// TIA Portal V18 export
// export: Created 2025-12-01T17:51:19.6025932Z, ExportSetting None, DisplayName Totally Integrated Automation Portal, DisplayVersion V18 Update 5, DisplayName TIA Portal Openness, DisplayVersion V18 Update 5, DisplayName TIA Portal Teamcenter Gateway, DisplayVersion V18, DisplayName TIA Portal Version Control Interface, DisplayVersion V18, DisplayName STEP 7 Professional, DisplayVersion V18 Update 5, DisplayName STEP 7 Safety, DisplayVersion V18, DisplayName WinCC Professional, DisplayVersion V18 Update 5
FUNCTION "Motorr" : Void   // FC3100, LAD
{ S7_Optimized_Access := 'TRUE' }
// stored: AutoNumber false, SetENOAutomatically false
   VAR_TEMP   // added for the SCL form of the ladder/FBD networks
      _w1 : Bool;
      _w2 : Bool;
   END_VAR
BEGIN

REGION Network 1: H-shaftLifting_Motor
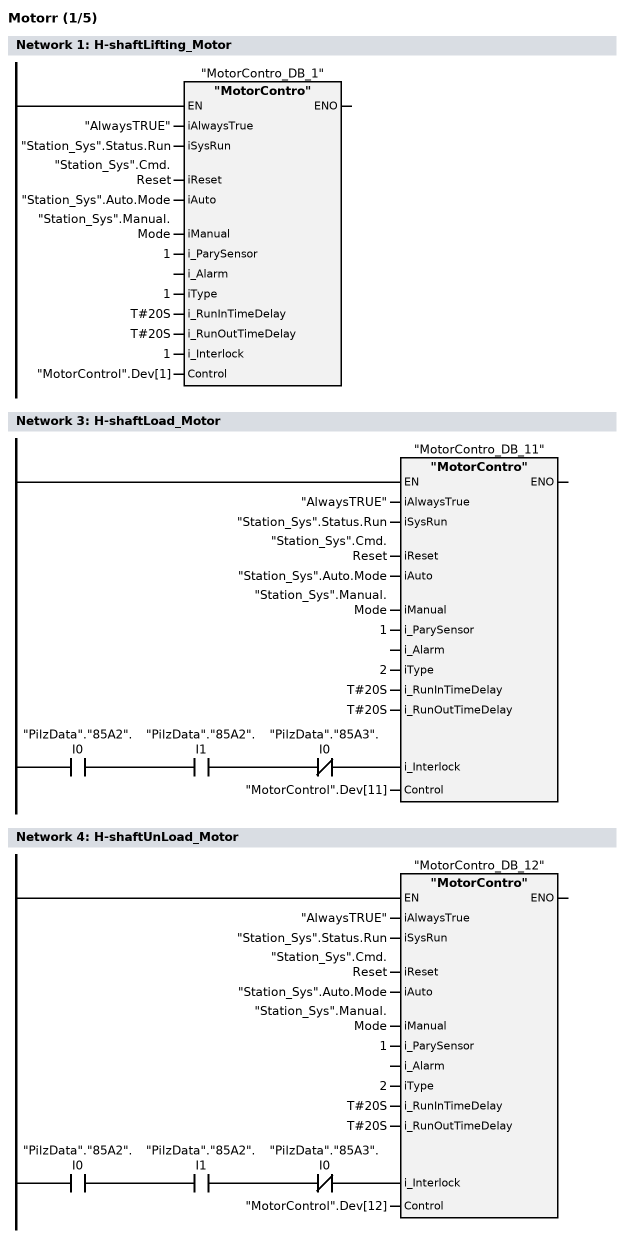
   RUNG wire#powerrail
      "MotorContro_DB_1"(iAlwaysTrue := "AlwaysTRUE", iSysRun := "Station_Sys".Status.Run, iReset := "Station_Sys".Cmd.Reset, iAuto := "Station_Sys".Auto.Mode, iManual := "Station_Sys".Manual.Mode, i_ParySensor := 1, i_Alarm :=, iType := 1, i_RunInTimeDelay := T#20S, i_RunOutTimeDelay := T#20S, i_Interlock := 1, Control := "MotorControl".Dev[1])
   END_RUNG
   // the same network as SCL:
   "MotorContro_DB_1"(iAlwaysTrue := "AlwaysTRUE",   // "MotorContro"
                      iSysRun := "Station_Sys".Status.Run,
                      iReset := "Station_Sys".Cmd.Reset,
                      iAuto := "Station_Sys".Auto.Mode,
                      iManual := "Station_Sys".Manual.Mode,
                      i_ParySensor := 1,
                      iType := 1,
                      i_RunInTimeDelay := T#20S,
                      i_RunOutTimeDelay := T#20S,
                      i_Interlock := 1,
                      Control := "MotorControl".Dev[1]);
END_REGION

REGION Network 2 (SCL): H-shaftLifting_Motor_OutPut
   "oH-shaftLifting_Start" := "MotorControl".Dev[1].OutControl.o_Start;
   "oH-shaftLifting_CCWStart" := "MotorControl".Dev[1].OutControl.o_CCWStart ;
   "oH-shaftLifting_SpeedChange" := "MotorControl".Dev[1].OutControl.o_SpeedChanged;
END_REGION

REGION Network 3: H-shaftLoad_Motor
   RUNG wire#powerrail
      "MotorContro_DB_11"(i_Interlock := wire#w1, iAlwaysTrue := "AlwaysTRUE", iSysRun := "Station_Sys".Status.Run, iReset := "Station_Sys".Cmd.Reset, iAuto := "Station_Sys".Auto.Mode, iManual := "Station_Sys".Manual.Mode, i_ParySensor := 1, i_Alarm :=, iType := 2, i_RunInTimeDelay := T#20S, i_RunOutTimeDelay := T#20S, Control := "MotorControl".Dev[11])
   END_RUNG
   RUNG wire#powerrail
      Contact( "PilzData"."85A2".I0 )
      Contact( "PilzData"."85A2".I1 )
      I_Contact( "PilzData"."85A3".I0 )
   END_RUNG wire#w1
   // the same network as SCL:
   "MotorContro_DB_11"(iAlwaysTrue := "AlwaysTRUE",   // "MotorContro"
                       iSysRun := "Station_Sys".Status.Run,
                       iReset := "Station_Sys".Cmd.Reset,
                       iAuto := "Station_Sys".Auto.Mode,
                       iManual := "Station_Sys".Manual.Mode,
                       i_ParySensor := 1,
                       iType := 2,
                       i_RunInTimeDelay := T#20S,
                       i_RunOutTimeDelay := T#20S,
                       i_Interlock := "PilzData"."85A2".I0 AND "PilzData"."85A2".I1 AND NOT "PilzData"."85A3".I0,
                       Control := "MotorControl".Dev[11]);
END_REGION

REGION Network 4: H-shaftUnLoad_Motor
   RUNG wire#powerrail
      "MotorContro_DB_12"(i_Interlock := wire#w1, iAlwaysTrue := "AlwaysTRUE", iSysRun := "Station_Sys".Status.Run, iReset := "Station_Sys".Cmd.Reset, iAuto := "Station_Sys".Auto.Mode, iManual := "Station_Sys".Manual.Mode, i_ParySensor := 1, i_Alarm :=, iType := 2, i_RunInTimeDelay := T#20S, i_RunOutTimeDelay := T#20S, Control := "MotorControl".Dev[12])
   END_RUNG
   RUNG wire#powerrail
      Contact( "PilzData"."85A2".I0 )
      Contact( "PilzData"."85A2".I1 )
      I_Contact( "PilzData"."85A3".I0 )
   END_RUNG wire#w1
   // the same network as SCL:
   "MotorContro_DB_12"(iAlwaysTrue := "AlwaysTRUE",   // "MotorContro"
                       iSysRun := "Station_Sys".Status.Run,
                       iReset := "Station_Sys".Cmd.Reset,
                       iAuto := "Station_Sys".Auto.Mode,
                       iManual := "Station_Sys".Manual.Mode,
                       i_ParySensor := 1,
                       iType := 2,
                       i_RunInTimeDelay := T#20S,
                       i_RunOutTimeDelay := T#20S,
                       i_Interlock := "PilzData"."85A2".I0 AND "PilzData"."85A2".I1 AND NOT "PilzData"."85A3".I0,
                       Control := "MotorControl".Dev[12]);
END_REGION

REGION Network 5 (SCL): H-shaftLifting_Motor_OutPut / H-shaftLoad_Motor_OutPut
   "oH-shaftLoading_CW" := "MotorControl".Dev[11].OutControl.o_Start;
   "oH-shaftLoading_CCW" := "MotorControl".Dev[11].OutControl.o_CCWStart OR ("Station_Sys".Auto.Mode AND "AutoProcessControl".Global.H.EmptyPallet);

   "oH-shaftTake_CW" := "MotorControl".Dev[12].OutControl.o_Start;
END_REGION

REGION Network 6: Auto MotorStop
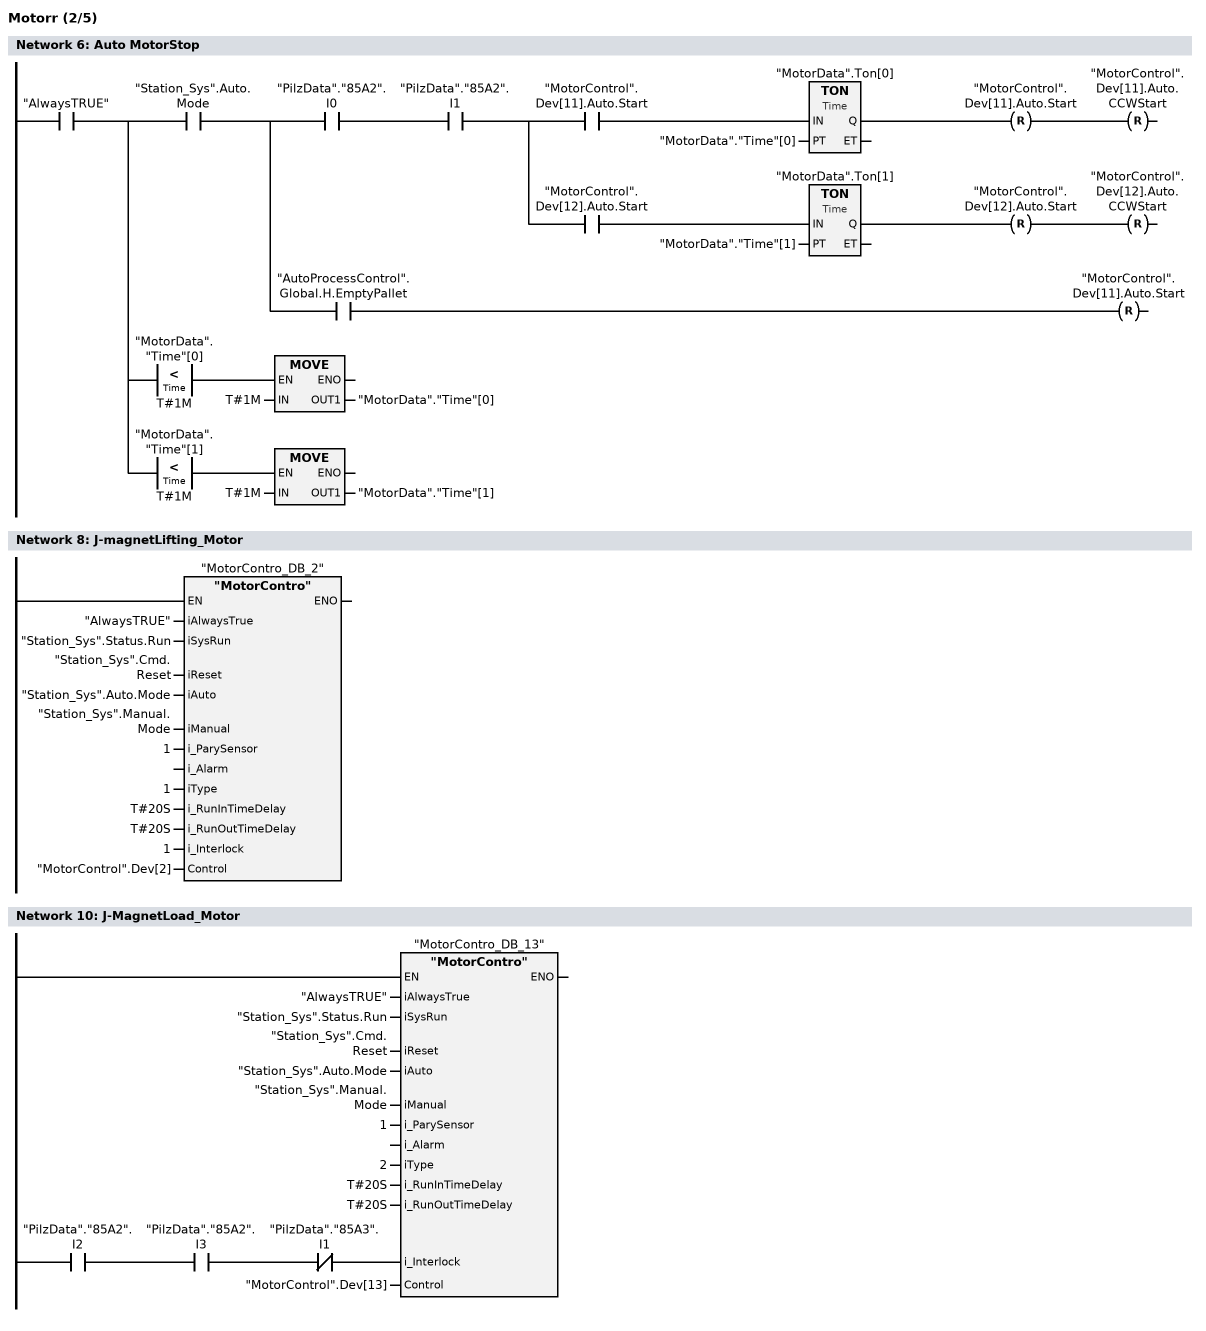
   RUNG wire#powerrail
      Contact( "AlwaysTRUE" )
      wire#w1
      Contact( "Station_Sys".Auto.Mode )
      wire#w2
      Contact( "PilzData"."85A2".I0 )
      Contact( "PilzData"."85A2".I1 )
      wire#w3
      Contact( "MotorControl".Dev[11].Auto.Start )
      { S7_Templates := "time_type := Time" } "MotorData".Ton[0].TON(pt := "MotorData"."Time"[0], et =>)
      R_Coil( "MotorControl".Dev[11].Auto.Start )
      R_Coil( "MotorControl".Dev[11].Auto.CCWStart )
   END_RUNG
   RUNG wire#w3
      Contact( "MotorControl".Dev[12].Auto.Start )
      { S7_Templates := "time_type := Time" } "MotorData".Ton[1].TON(pt := "MotorData"."Time"[1], et =>)
      R_Coil( "MotorControl".Dev[12].Auto.Start )
      R_Coil( "MotorControl".Dev[12].Auto.CCWStart )
   END_RUNG
   RUNG wire#w2
      Contact( "AutoProcessControl".Global.H.EmptyPallet )
      R_Coil( "MotorControl".Dev[11].Auto.Start )
   END_RUNG
   RUNG wire#w1
      { S7_Templates := "SrcType := Time" } LT_Contact(in1 := "MotorData"."Time"[0], in2 := T#1M)
      Move(in := T#1M, out1 => "MotorData"."Time"[0])
   END_RUNG
   RUNG wire#w1
      { S7_Templates := "SrcType := Time" } LT_Contact(in1 := "MotorData"."Time"[1], in2 := T#1M)
      Move(in := T#1M, out1 => "MotorData"."Time"[1])
   END_RUNG
   // the same network as SCL:
   #_w1 := "AlwaysTRUE" AND "Station_Sys".Auto.Mode;
   #_w2 := #_w1 AND "PilzData"."85A2".I0 AND "PilzData"."85A2".I1;
   "MotorData".Ton[0].TON(IN := #_w2 AND "MotorControl".Dev[11].Auto.Start, PT := "MotorData"."Time"[0]);
   IF "MotorData".Ton[0].Q THEN
       "MotorControl".Dev[11].Auto.Start := FALSE;
       "MotorControl".Dev[11].Auto.CCWStart := FALSE;
   END_IF;
   "MotorData".Ton[1].TON(IN := #_w2 AND "MotorControl".Dev[12].Auto.Start, PT := "MotorData"."Time"[1]);
   IF "MotorData".Ton[1].Q THEN
       "MotorControl".Dev[12].Auto.Start := FALSE;
       "MotorControl".Dev[12].Auto.CCWStart := FALSE;
   END_IF;
   IF #_w1 AND "AutoProcessControl".Global.H.EmptyPallet THEN
       "MotorControl".Dev[11].Auto.Start := FALSE;
   END_IF;
   IF "AlwaysTRUE" AND ("MotorData"."Time"[0] < T#1M) THEN "MotorData"."Time"[0] := T#1M; END_IF;
   IF "AlwaysTRUE" AND ("MotorData"."Time"[1] < T#1M) THEN "MotorData"."Time"[1] := T#1M; END_IF;
END_REGION

REGION Network 8: J-magnetLifting_Motor
   RUNG wire#powerrail
      "MotorContro_DB_2"(iAlwaysTrue := "AlwaysTRUE", iSysRun := "Station_Sys".Status.Run, iReset := "Station_Sys".Cmd.Reset, iAuto := "Station_Sys".Auto.Mode, iManual := "Station_Sys".Manual.Mode, i_ParySensor := 1, i_Alarm :=, iType := 1, i_RunInTimeDelay := T#20S, i_RunOutTimeDelay := T#20S, i_Interlock := 1, Control := "MotorControl".Dev[2])
   END_RUNG
   // the same network as SCL:
   "MotorContro_DB_2"(iAlwaysTrue := "AlwaysTRUE",   // "MotorContro"
                      iSysRun := "Station_Sys".Status.Run,
                      iReset := "Station_Sys".Cmd.Reset,
                      iAuto := "Station_Sys".Auto.Mode,
                      iManual := "Station_Sys".Manual.Mode,
                      i_ParySensor := 1,
                      iType := 1,
                      i_RunInTimeDelay := T#20S,
                      i_RunOutTimeDelay := T#20S,
                      i_Interlock := 1,
                      Control := "MotorControl".Dev[2]);
END_REGION

REGION Network 9 (SCL): J-magnetLifting_Motor_OutPut
   "oJ-magnetLifting_Start" := "MotorControl".Dev[2].OutControl.o_Start;
   "oJ-magnetLifting_CCWStart" := "MotorControl".Dev[2].OutControl.o_CCWStart;
   "oJ-magnetLifting_SpeedChange" := "MotorControl".Dev[2].OutControl.o_SpeedChanged;
END_REGION

REGION Network 10: J-MagnetLoad_Motor
   RUNG wire#powerrail
      "MotorContro_DB_13"(i_Interlock := wire#w1, iAlwaysTrue := "AlwaysTRUE", iSysRun := "Station_Sys".Status.Run, iReset := "Station_Sys".Cmd.Reset, iAuto := "Station_Sys".Auto.Mode, iManual := "Station_Sys".Manual.Mode, i_ParySensor := 1, i_Alarm :=, iType := 2, i_RunInTimeDelay := T#20S, i_RunOutTimeDelay := T#20S, Control := "MotorControl".Dev[13])
   END_RUNG
   RUNG wire#powerrail
      Contact( "PilzData"."85A2".I2 )
      Contact( "PilzData"."85A2".I3 )
      I_Contact( "PilzData"."85A3".I1 )
   END_RUNG wire#w1
   // the same network as SCL:
   "MotorContro_DB_13"(iAlwaysTrue := "AlwaysTRUE",   // "MotorContro"
                       iSysRun := "Station_Sys".Status.Run,
                       iReset := "Station_Sys".Cmd.Reset,
                       iAuto := "Station_Sys".Auto.Mode,
                       iManual := "Station_Sys".Manual.Mode,
                       i_ParySensor := 1,
                       iType := 2,
                       i_RunInTimeDelay := T#20S,
                       i_RunOutTimeDelay := T#20S,
                       i_Interlock := "PilzData"."85A2".I2 AND "PilzData"."85A2".I3 AND NOT "PilzData"."85A3".I1,
                       Control := "MotorControl".Dev[13]);
END_REGION

REGION Network 11: J-MagnetUnLoad_Motor
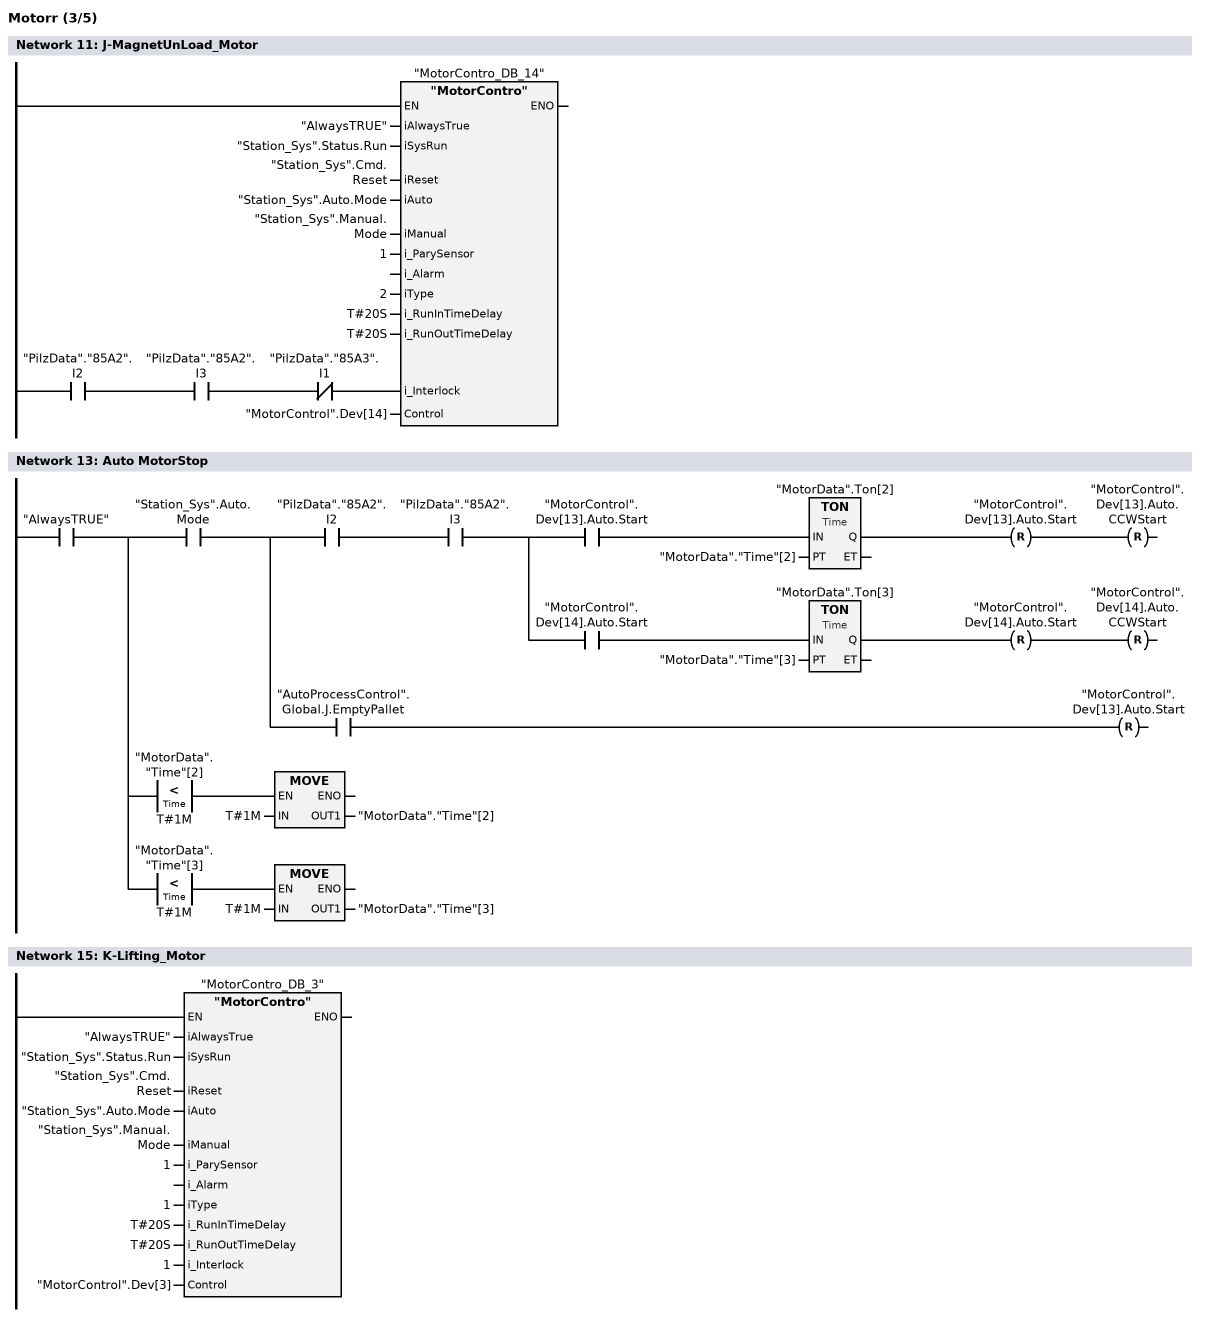
   RUNG wire#powerrail
      "MotorContro_DB_14"(i_Interlock := wire#w1, iAlwaysTrue := "AlwaysTRUE", iSysRun := "Station_Sys".Status.Run, iReset := "Station_Sys".Cmd.Reset, iAuto := "Station_Sys".Auto.Mode, iManual := "Station_Sys".Manual.Mode, i_ParySensor := 1, i_Alarm :=, iType := 2, i_RunInTimeDelay := T#20S, i_RunOutTimeDelay := T#20S, Control := "MotorControl".Dev[14])
   END_RUNG
   RUNG wire#powerrail
      Contact( "PilzData"."85A2".I2 )
      Contact( "PilzData"."85A2".I3 )
      I_Contact( "PilzData"."85A3".I1 )
   END_RUNG wire#w1
   // the same network as SCL:
   "MotorContro_DB_14"(iAlwaysTrue := "AlwaysTRUE",   // "MotorContro"
                       iSysRun := "Station_Sys".Status.Run,
                       iReset := "Station_Sys".Cmd.Reset,
                       iAuto := "Station_Sys".Auto.Mode,
                       iManual := "Station_Sys".Manual.Mode,
                       i_ParySensor := 1,
                       iType := 2,
                       i_RunInTimeDelay := T#20S,
                       i_RunOutTimeDelay := T#20S,
                       i_Interlock := "PilzData"."85A2".I2 AND "PilzData"."85A2".I3 AND NOT "PilzData"."85A3".I1,
                       Control := "MotorControl".Dev[14]);
END_REGION

REGION Network 12 (SCL): H-shaftLifting_Motor_OutPut / J-Magnet_Motor_OutPut
   "J-magnet Loading _CW" := "MotorControl".Dev[13].OutControl.o_Start;
   "J-magnet Loading _CCW" := "MotorControl".Dev[13].OutControl.o_CCWStart OR ("Station_Sys".Auto.Mode AND "AutoProcessControl".Global.J.EmptyPallet);

   "J-magnet Take _CW" := "MotorControl".Dev[14].OutControl.o_Start;
END_REGION

REGION Network 13: Auto MotorStop
   RUNG wire#powerrail
      Contact( "AlwaysTRUE" )
      wire#w1
      Contact( "Station_Sys".Auto.Mode )
      wire#w2
      Contact( "PilzData"."85A2".I2 )
      Contact( "PilzData"."85A2".I3 )
      wire#w3
      Contact( "MotorControl".Dev[13].Auto.Start )
      { S7_Templates := "time_type := Time" } "MotorData".Ton[2].TON(pt := "MotorData"."Time"[2], et =>)
      R_Coil( "MotorControl".Dev[13].Auto.Start )
      R_Coil( "MotorControl".Dev[13].Auto.CCWStart )
   END_RUNG
   RUNG wire#w3
      Contact( "MotorControl".Dev[14].Auto.Start )
      { S7_Templates := "time_type := Time" } "MotorData".Ton[3].TON(pt := "MotorData"."Time"[3], et =>)
      R_Coil( "MotorControl".Dev[14].Auto.Start )
      R_Coil( "MotorControl".Dev[14].Auto.CCWStart )
   END_RUNG
   RUNG wire#w2
      Contact( "AutoProcessControl".Global.J.EmptyPallet )
      R_Coil( "MotorControl".Dev[13].Auto.Start )
   END_RUNG
   RUNG wire#w1
      { S7_Templates := "SrcType := Time" } LT_Contact(in1 := "MotorData"."Time"[2], in2 := T#1M)
      Move(in := T#1M, out1 => "MotorData"."Time"[2])
   END_RUNG
   RUNG wire#w1
      { S7_Templates := "SrcType := Time" } LT_Contact(in1 := "MotorData"."Time"[3], in2 := T#1M)
      Move(in := T#1M, out1 => "MotorData"."Time"[3])
   END_RUNG
   // the same network as SCL:
   #_w1 := "AlwaysTRUE" AND "Station_Sys".Auto.Mode;
   #_w2 := #_w1 AND "PilzData"."85A2".I2 AND "PilzData"."85A2".I3;
   "MotorData".Ton[2].TON(IN := #_w2 AND "MotorControl".Dev[13].Auto.Start, PT := "MotorData"."Time"[2]);
   IF "MotorData".Ton[2].Q THEN
       "MotorControl".Dev[13].Auto.Start := FALSE;
       "MotorControl".Dev[13].Auto.CCWStart := FALSE;
   END_IF;
   "MotorData".Ton[3].TON(IN := #_w2 AND "MotorControl".Dev[14].Auto.Start, PT := "MotorData"."Time"[3]);
   IF "MotorData".Ton[3].Q THEN
       "MotorControl".Dev[14].Auto.Start := FALSE;
       "MotorControl".Dev[14].Auto.CCWStart := FALSE;
   END_IF;
   IF #_w1 AND "AutoProcessControl".Global.J.EmptyPallet THEN
       "MotorControl".Dev[13].Auto.Start := FALSE;
   END_IF;
   IF "AlwaysTRUE" AND ("MotorData"."Time"[2] < T#1M) THEN "MotorData"."Time"[2] := T#1M; END_IF;
   IF "AlwaysTRUE" AND ("MotorData"."Time"[3] < T#1M) THEN "MotorData"."Time"[3] := T#1M; END_IF;
END_REGION

REGION Network 15: K-Lifting_Motor
   RUNG wire#powerrail
      "MotorContro_DB_3"(iAlwaysTrue := "AlwaysTRUE", iSysRun := "Station_Sys".Status.Run, iReset := "Station_Sys".Cmd.Reset, iAuto := "Station_Sys".Auto.Mode, iManual := "Station_Sys".Manual.Mode, i_ParySensor := 1, i_Alarm :=, iType := 1, i_RunInTimeDelay := T#20S, i_RunOutTimeDelay := T#20S, i_Interlock := 1, Control := "MotorControl".Dev[3])
   END_RUNG
   // the same network as SCL:
   "MotorContro_DB_3"(iAlwaysTrue := "AlwaysTRUE",   // "MotorContro"
                      iSysRun := "Station_Sys".Status.Run,
                      iReset := "Station_Sys".Cmd.Reset,
                      iAuto := "Station_Sys".Auto.Mode,
                      iManual := "Station_Sys".Manual.Mode,
                      i_ParySensor := 1,
                      iType := 1,
                      i_RunInTimeDelay := T#20S,
                      i_RunOutTimeDelay := T#20S,
                      i_Interlock := 1,
                      Control := "MotorControl".Dev[3]);
END_REGION

REGION Network 16 (SCL): K-Lifting_Motor_OutPut
   "oK-Lifting3_Start" := "MotorControl".Dev[3].OutControl.o_Start;
   "oK-Lifting3_CCWStart" := "MotorControl".Dev[3].OutControl.o_CCWStart;
   "oK-Lifting3_SpeedChange" := "MotorControl".Dev[3].OutControl.o_SpeedChanged;
END_REGION

REGION Network 17: K-ReserveLoad_Motor
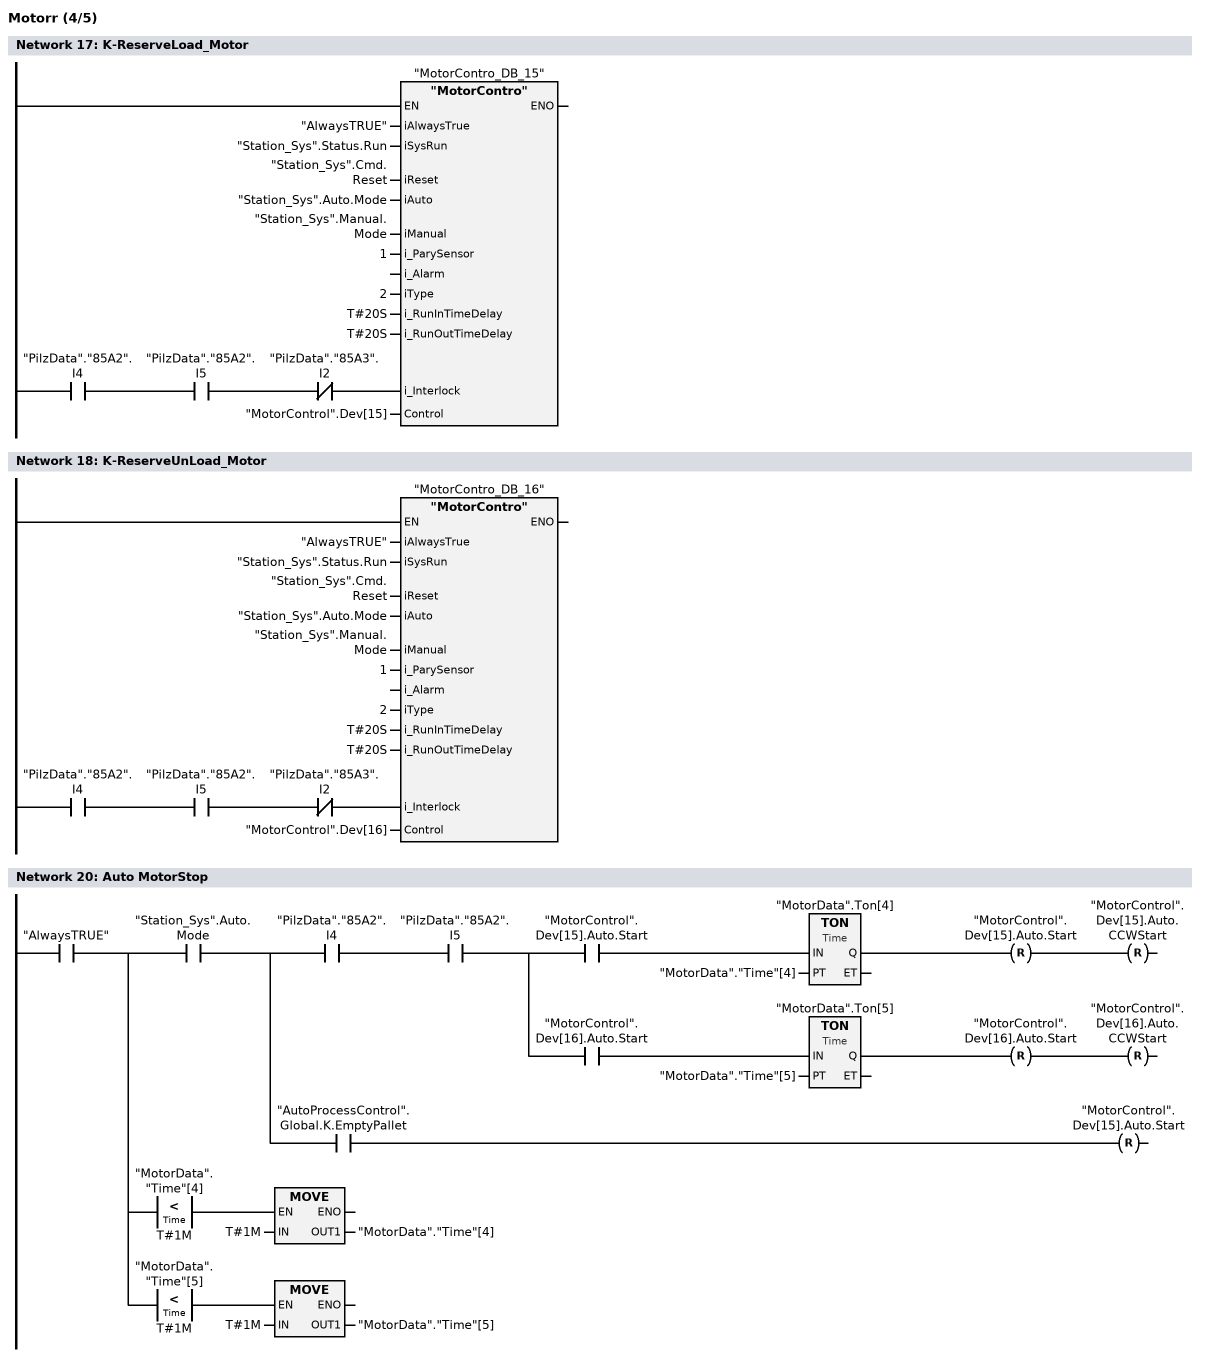
   RUNG wire#powerrail
      "MotorContro_DB_15"(i_Interlock := wire#w1, iAlwaysTrue := "AlwaysTRUE", iSysRun := "Station_Sys".Status.Run, iReset := "Station_Sys".Cmd.Reset, iAuto := "Station_Sys".Auto.Mode, iManual := "Station_Sys".Manual.Mode, i_ParySensor := 1, i_Alarm :=, iType := 2, i_RunInTimeDelay := T#20S, i_RunOutTimeDelay := T#20S, Control := "MotorControl".Dev[15])
   END_RUNG
   RUNG wire#powerrail
      Contact( "PilzData"."85A2".I4 )
      Contact( "PilzData"."85A2".I5 )
      I_Contact( "PilzData"."85A3".I2 )
   END_RUNG wire#w1
   // the same network as SCL:
   "MotorContro_DB_15"(iAlwaysTrue := "AlwaysTRUE",   // "MotorContro"
                       iSysRun := "Station_Sys".Status.Run,
                       iReset := "Station_Sys".Cmd.Reset,
                       iAuto := "Station_Sys".Auto.Mode,
                       iManual := "Station_Sys".Manual.Mode,
                       i_ParySensor := 1,
                       iType := 2,
                       i_RunInTimeDelay := T#20S,
                       i_RunOutTimeDelay := T#20S,
                       i_Interlock := "PilzData"."85A2".I4 AND "PilzData"."85A2".I5 AND NOT "PilzData"."85A3".I2,
                       Control := "MotorControl".Dev[15]);
END_REGION

REGION Network 18: K-ReserveUnLoad_Motor
   RUNG wire#powerrail
      "MotorContro_DB_16"(i_Interlock := wire#w1, iAlwaysTrue := "AlwaysTRUE", iSysRun := "Station_Sys".Status.Run, iReset := "Station_Sys".Cmd.Reset, iAuto := "Station_Sys".Auto.Mode, iManual := "Station_Sys".Manual.Mode, i_ParySensor := 1, i_Alarm :=, iType := 2, i_RunInTimeDelay := T#20S, i_RunOutTimeDelay := T#20S, Control := "MotorControl".Dev[16])
   END_RUNG
   RUNG wire#powerrail
      Contact( "PilzData"."85A2".I4 )
      Contact( "PilzData"."85A2".I5 )
      I_Contact( "PilzData"."85A3".I2 )
   END_RUNG wire#w1
   // the same network as SCL:
   "MotorContro_DB_16"(iAlwaysTrue := "AlwaysTRUE",   // "MotorContro"
                       iSysRun := "Station_Sys".Status.Run,
                       iReset := "Station_Sys".Cmd.Reset,
                       iAuto := "Station_Sys".Auto.Mode,
                       iManual := "Station_Sys".Manual.Mode,
                       i_ParySensor := 1,
                       iType := 2,
                       i_RunInTimeDelay := T#20S,
                       i_RunOutTimeDelay := T#20S,
                       i_Interlock := "PilzData"."85A2".I4 AND "PilzData"."85A2".I5 AND NOT "PilzData"."85A3".I2,
                       Control := "MotorControl".Dev[16]);
END_REGION

REGION Network 19 (SCL): H-shaftLifting_Motor_OutPut / K-Reserve_Motor_OutPut
   "K-Loading _CW" := "MotorControl".Dev[15].OutControl.o_Start;
   "K-Loading _CCW" := "MotorControl".Dev[15].OutControl.o_CCWStart OR ("Station_Sys".Auto.Mode AND "AutoProcessControl".Global.K.EmptyPallet);

   "K-Take _CW" := "MotorControl".Dev[16].OutControl.o_Start;
END_REGION

REGION Network 20: Auto MotorStop
   RUNG wire#powerrail
      Contact( "AlwaysTRUE" )
      wire#w1
      Contact( "Station_Sys".Auto.Mode )
      wire#w2
      Contact( "PilzData"."85A2".I4 )
      Contact( "PilzData"."85A2".I5 )
      wire#w3
      Contact( "MotorControl".Dev[15].Auto.Start )
      { S7_Templates := "time_type := Time" } "MotorData".Ton[4].TON(pt := "MotorData"."Time"[4], et =>)
      R_Coil( "MotorControl".Dev[15].Auto.Start )
      R_Coil( "MotorControl".Dev[15].Auto.CCWStart )
   END_RUNG
   RUNG wire#w3
      Contact( "MotorControl".Dev[16].Auto.Start )
      { S7_Templates := "time_type := Time" } "MotorData".Ton[5].TON(pt := "MotorData"."Time"[5], et =>)
      R_Coil( "MotorControl".Dev[16].Auto.Start )
      R_Coil( "MotorControl".Dev[16].Auto.CCWStart )
   END_RUNG
   RUNG wire#w2
      Contact( "AutoProcessControl".Global.K.EmptyPallet )
      R_Coil( "MotorControl".Dev[15].Auto.Start )
   END_RUNG
   RUNG wire#w1
      { S7_Templates := "SrcType := Time" } LT_Contact(in1 := "MotorData"."Time"[4], in2 := T#1M)
      Move(in := T#1M, out1 => "MotorData"."Time"[4])
   END_RUNG
   RUNG wire#w1
      { S7_Templates := "SrcType := Time" } LT_Contact(in1 := "MotorData"."Time"[5], in2 := T#1M)
      Move(in := T#1M, out1 => "MotorData"."Time"[5])
   END_RUNG
   // the same network as SCL:
   #_w1 := "AlwaysTRUE" AND "Station_Sys".Auto.Mode;
   #_w2 := #_w1 AND "PilzData"."85A2".I4 AND "PilzData"."85A2".I5;
   "MotorData".Ton[4].TON(IN := #_w2 AND "MotorControl".Dev[15].Auto.Start, PT := "MotorData"."Time"[4]);
   IF "MotorData".Ton[4].Q THEN
       "MotorControl".Dev[15].Auto.Start := FALSE;
       "MotorControl".Dev[15].Auto.CCWStart := FALSE;
   END_IF;
   "MotorData".Ton[5].TON(IN := #_w2 AND "MotorControl".Dev[16].Auto.Start, PT := "MotorData"."Time"[5]);
   IF "MotorData".Ton[5].Q THEN
       "MotorControl".Dev[16].Auto.Start := FALSE;
       "MotorControl".Dev[16].Auto.CCWStart := FALSE;
   END_IF;
   IF #_w1 AND "AutoProcessControl".Global.K.EmptyPallet THEN
       "MotorControl".Dev[15].Auto.Start := FALSE;
   END_IF;
   IF "AlwaysTRUE" AND ("MotorData"."Time"[4] < T#1M) THEN "MotorData"."Time"[4] := T#1M; END_IF;
   IF "AlwaysTRUE" AND ("MotorData"."Time"[5] < T#1M) THEN "MotorData"."Time"[5] := T#1M; END_IF;
END_REGION

REGION Network 22: L-Unloading_Motor
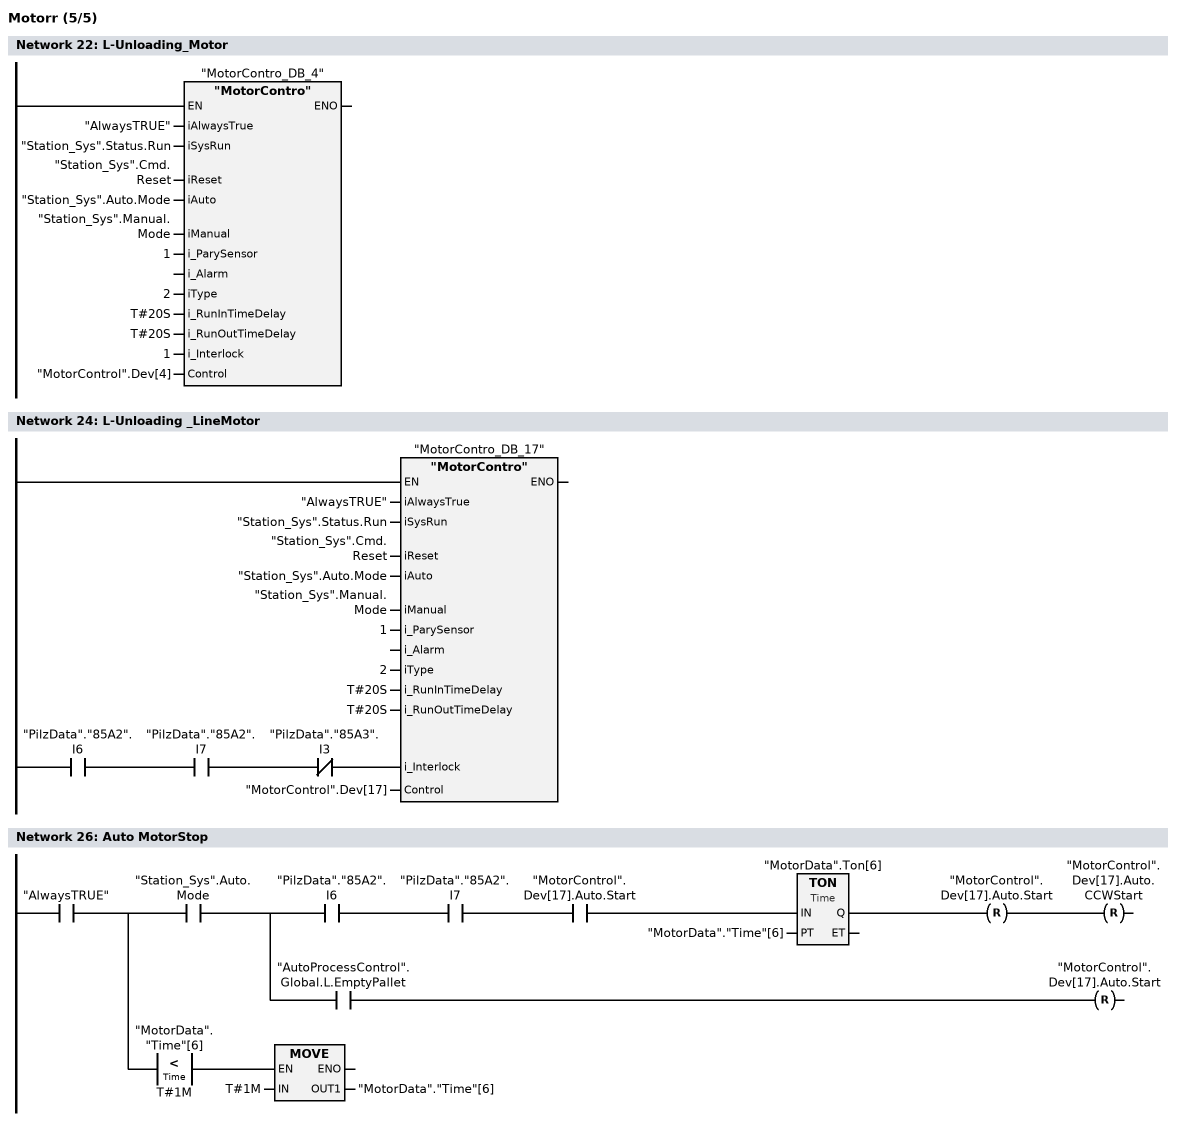
   RUNG wire#powerrail
      "MotorContro_DB_4"(iAlwaysTrue := "AlwaysTRUE", iSysRun := "Station_Sys".Status.Run, iReset := "Station_Sys".Cmd.Reset, iAuto := "Station_Sys".Auto.Mode, iManual := "Station_Sys".Manual.Mode, i_ParySensor := 1, i_Alarm :=, iType := 2, i_RunInTimeDelay := T#20S, i_RunOutTimeDelay := T#20S, i_Interlock := 1, Control := "MotorControl".Dev[4])
   END_RUNG
   // the same network as SCL:
   "MotorContro_DB_4"(iAlwaysTrue := "AlwaysTRUE",   // "MotorContro"
                      iSysRun := "Station_Sys".Status.Run,
                      iReset := "Station_Sys".Cmd.Reset,
                      iAuto := "Station_Sys".Auto.Mode,
                      iManual := "Station_Sys".Manual.Mode,
                      i_ParySensor := 1,
                      iType := 2,
                      i_RunInTimeDelay := T#20S,
                      i_RunOutTimeDelay := T#20S,
                      i_Interlock := 1,
                      Control := "MotorControl".Dev[4]);
END_REGION

REGION Network 23 (SCL): L-Unloading_Motor_OutPut
   "oL-Unloading_CW" := "MotorControl".Dev[4].OutControl.o_Start;
   "oL-Unloading_CCW" := "MotorControl".Dev[4].OutControl.o_CCWStart;
END_REGION

REGION Network 24: L-Unloading _LineMotor
   RUNG wire#powerrail
      "MotorContro_DB_17"(i_Interlock := wire#w1, iAlwaysTrue := "AlwaysTRUE", iSysRun := "Station_Sys".Status.Run, iReset := "Station_Sys".Cmd.Reset, iAuto := "Station_Sys".Auto.Mode, iManual := "Station_Sys".Manual.Mode, i_ParySensor := 1, i_Alarm :=, iType := 2, i_RunInTimeDelay := T#20S, i_RunOutTimeDelay := T#20S, Control := "MotorControl".Dev[17])
   END_RUNG
   RUNG wire#powerrail
      Contact( "PilzData"."85A2".I6 )
      Contact( "PilzData"."85A2".I7 )
      I_Contact( "PilzData"."85A3".I3 )
   END_RUNG wire#w1
   // the same network as SCL:
   "MotorContro_DB_17"(iAlwaysTrue := "AlwaysTRUE",   // "MotorContro"
                       iSysRun := "Station_Sys".Status.Run,
                       iReset := "Station_Sys".Cmd.Reset,
                       iAuto := "Station_Sys".Auto.Mode,
                       iManual := "Station_Sys".Manual.Mode,
                       i_ParySensor := 1,
                       iType := 2,
                       i_RunInTimeDelay := T#20S,
                       i_RunOutTimeDelay := T#20S,
                       i_Interlock := "PilzData"."85A2".I6 AND "PilzData"."85A2".I7 AND NOT "PilzData"."85A3".I3,
                       Control := "MotorControl".Dev[17]);
END_REGION

REGION Network 25 (SCL): H-shaftLifting_Motor_OutPut / L-Unloading _LineMotor_OutPut
   "L-Unloading _LineMotor_CW" := "MotorControl".Dev[17].OutControl.o_Start;
   "L-Unloading _LineMotor_CCW" := "MotorControl".Dev[17].OutControl.o_CCWStart OR ("Station_Sys".Auto.Mode AND "AutoProcessControl".Global.L.EmptyPallet);
END_REGION

REGION Network 26: Auto MotorStop
   RUNG wire#powerrail
      Contact( "AlwaysTRUE" )
      wire#w1
      Contact( "Station_Sys".Auto.Mode )
      wire#w2
      Contact( "PilzData"."85A2".I6 )
      Contact( "PilzData"."85A2".I7 )
      Contact( "MotorControl".Dev[17].Auto.Start )
      { S7_Templates := "time_type := Time" } "MotorData".Ton[6].TON(pt := "MotorData"."Time"[6], et =>)
      R_Coil( "MotorControl".Dev[17].Auto.Start )
      R_Coil( "MotorControl".Dev[17].Auto.CCWStart )
   END_RUNG
   RUNG wire#w2
      Contact( "AutoProcessControl".Global.L.EmptyPallet )
      R_Coil( "MotorControl".Dev[17].Auto.Start )
   END_RUNG
   RUNG wire#w1
      { S7_Templates := "SrcType := Time" } LT_Contact(in1 := "MotorData"."Time"[6], in2 := T#1M)
      Move(in := T#1M, out1 => "MotorData"."Time"[6])
   END_RUNG
   // the same network as SCL:
   #_w1 := "AlwaysTRUE" AND "Station_Sys".Auto.Mode;
   "MotorData".Ton[6].TON(IN := #_w1 AND "PilzData"."85A2".I6 AND "PilzData"."85A2".I7 AND "MotorControl".Dev[17].Auto.Start,
                          PT := "MotorData"."Time"[6]);
   IF "MotorData".Ton[6].Q THEN
       "MotorControl".Dev[17].Auto.Start := FALSE;
       "MotorControl".Dev[17].Auto.CCWStart := FALSE;
   END_IF;
   IF #_w1 AND "AutoProcessControl".Global.L.EmptyPallet THEN
       "MotorControl".Dev[17].Auto.Start := FALSE;
   END_IF;
   IF "AlwaysTRUE" AND ("MotorData"."Time"[6] < T#1M) THEN "MotorData"."Time"[6] := T#1M; END_IF;
END_REGION
END_FUNCTION
